// TIA Portal project "Projet_final_groupe_01" (V15.1)

(* hardware
DEVICE "Station S71500/ET200MP_1"  S7-1500 station
   slot 0: "Châssis_0"  Rack  6ES7 590-1***0-0AA0
   slot 1: "PLC_1"  CPU 1513-1 PN  6ES7 513-1AL00-0AB0  V1.7
      slot 3: "Ecran CPU_1"  6ES7591-1AA00-0AA0
   slot 2: "DI 32x24VDC HF_1"  DI 32x24VDC HF  6ES7 521-1BL00-0AB0  V2.0
   slot 3: "DQ 32x24VDC/0.5A ST_1"  DQ 32x24VDC/0.5A ST  6ES7 522-1BL00-0AB0  V2.0
DEVICE "Appareil GSD_1"  GSD.Device.PN
   slot 0: "Châssis"  Rack  V1.0
   slot 0: "PNET-Anybus"  DSQC688  ABCC-PRT  V1.12
      slot 0: "PROFINET Anybus"  PROFINET Anybus  ABCC-PRT  V1.12
      slot 1: "Interface"  Interface
         slot 1: "Port 1"  Port 1
   slot 1: "Input 64 byte_1"  Input 64 byte  V1.0
      slot 0: "Input 64 byte"  Input 64 byte
   slot 2: "Output 64 byte_1"  Output 64 byte  V1.0
      slot 0: "Output 64 byte"  Output 64 byte
DEVICE "Appareil GSD_2"  GSD.Device.PN
   slot 0: "Châssis"  Rack  V1.0
   slot 0: "AL1100"  AL1100  AL1100
      slot 0: "AL1100"  AL1100
      slot 1: "X1"  X1
         slot 1: "Port 1"  Port 1
         slot 2: "Port 2"  Port 2
      slot 1: "4 Ports_1"  4 Ports  AL1100
         slot 0: "IO-Link Master"  IO-Link Master
   slot 1: "IO-Link In  2 Byte + PQI"  IO-Link In  2 Byte + PQI
   slot 2: "Disabled"  Disabled
   slot 3: "Disabled_1"  Disabled
   slot 4: "Disabled_2"  Disabled
*)

// ===== PLC "PLC_1"  CPU 1513-1 PN =====

VAR_GLOBAL   // PLC tag table "Table de variables standard"
   "Sécurité_active" AT %M5.0 : Bool;
   "Marche_cycle" AT %M5.1 : Bool;
   "System_Byte" AT %MB1 : Byte;
   "FirstScan" AT %M1.0 : Bool;
   "DiagStatusUpdate" AT %M1.1 : Bool;
   "AlwaysTRUE" AT %M1.2 : Bool;
   "AlwaysFALSE" AT %M1.3 : Bool;
   "Clock_Byte" AT %MB0 : Byte;
   "Clock_10Hz" AT %M0.0 : Bool;
   "Clock_5Hz" AT %M0.1 : Bool;
   "Clock_2.5Hz" AT %M0.2 : Bool;
   "Clock_2Hz" AT %M0.3 : Bool;
   "Clock_1.25Hz" AT %M0.4 : Bool;
   "Clock_1Hz" AT %M0.5 : Bool;
   "Clock_0.625Hz" AT %M0.6 : Bool;
   "Clock_0.5Hz" AT %M0.7 : Bool;
END_VAR

VAR_GLOBAL   // PLC tag table "Table de variables standard_1"
   "Sécurité_active(1)" AT %M5.0 : Bool;
   "Marche_cycle(1)" AT %M5.1 : Bool;
   "MDM_Local" AT %M5.2 : Bool;
   "MDM_Distant" AT %M5.3 : Bool;
   "MDM_Maintenance" AT %M5.4 : Bool;
   "Demande_arret_propre" AT %M5.5 : Bool;
END_VAR

VAR_GLOBAL CONSTANT   // PLC tag table "Table de variables standard_1"
   "Aucun(e)(1)" : Pip := 65535;
   "Mise à jour automatique(1)" : Pip := 0;
   "MIP 1(1)" : Pip := 1;
   "MIP 2(1)" : Pip := 2;
   "MIP 3(1)" : Pip := 3;
   "MIP 4(1)" : Pip := 4;
   "MIP 5(1)" : Pip := 5;
   "MIP 6(1)" : Pip := 6;
   "MIP 7(1)" : Pip := 7;
   "MIP 8(1)" : Pip := 8;
   "MIP 9(1)" : Pip := 9;
   "MIP 10(1)" : Pip := 10;
   "MIP 11(1)" : Pip := 11;
   "MIP 12(1)" : Pip := 12;
   "MIP 13(1)" : Pip := 13;
   "MIP 14(1)" : Pip := 14;
   "MIP 15(1)" : Pip := 15;
   "MIP 16(1)" : Pip := 16;
   "MIP 17(1)" : Pip := 17;
   "MIP 18(1)" : Pip := 18;
   "MIP 19(1)" : Pip := 19;
   "MIP 20(1)" : Pip := 20;
   "MIP 21(1)" : Pip := 21;
   "MIP 22(1)" : Pip := 22;
   "MIP 23(1)" : Pip := 23;
   "MIP 24(1)" : Pip := 24;
   "MIP 25(1)" : Pip := 25;
   "MIP 26(1)" : Pip := 26;
   "MIP 27(1)" : Pip := 27;
   "MIP 28(1)" : Pip := 28;
   "MIP 29(1)" : Pip := 29;
   "MIP 30(1)" : Pip := 30;
   "MIP 31(1)" : Pip := 31;
   "MIP OB Servo(1)" : Pip := 32768;
   "Local(1)" : Hw_SubModule := 49;
   "Local~Common(1)" : Hw_SubModule := 50;
   "Local~Device(1)" : Hw_Device := 32;
   "Local~Configuration(1)" : Hw_SubModule := 33;
   "Local~Display(1)" : Hw_SubModule := 54;
   "Local~MC(1)" : Hw_SubModule := 51;
   "Local~Exec(1)" : Hw_SubModule := 52;
   "Local~Interface_PROFINET_1(1)" : Hw_Interface := 64;
   "Local~Interface_PROFINET_1~Port_1(1)" : Hw_Interface := 65;
   "Local~Interface_PROFINET_1~Port_2(1)" : Hw_Interface := 66;
   "Local~DI_32x24VDC_HF_1(1)" : Hw_SubModule := 257;
   "Local~DQ_32x24VDC_0_5A_ST_1(1)" : Hw_SubModule := 258;
   "OB_Main(1)" : OB_PCYCLE := 1;
   "Local~PROFINET_IO-System(1)" : Hw_IoSystem := 259;
   "AL1100~Proxy(1)" : Hw_SubModule := 266;
   "AL1100~IODevice(1)" : Hw_Device := 263;
   "AL1100~X1(1)" : Hw_Interface := 267;
   "AL1100~X1~Port_1(1)" : Hw_Interface := 260;
   "AL1100~X1~Port_2(1)" : Hw_Interface := 261;
   "AL1100~Head(1)" : Hw_SubModule := 262;
   "AL1100~4_Ports_1(1)" : Hw_SubModule := 264;
   "PNET-Anybus~Proxy(1)" : Hw_SubModule := 270;
   "PNET-Anybus~IODevice(1)" : Hw_Device := 268;
   "PNET-Anybus~Interface(1)" : Hw_Interface := 271;
   "PNET-Anybus~Interface~Port_1(1)" : Hw_Interface := 272;
   "PNET-Anybus~Head(1)" : Hw_SubModule := 273;
   "PNET-Anybus~Input_64_byte_1(1)" : Hw_SubModule := 274;
   "PNET-Anybus~Output_64_byte_1(1)" : Hw_SubModule := 275;
   "AL1100~4_Ports_1_1(1)" : Hw_SubModule := 276;
   "AL1100~4_Ports_1~IO-Link_In__2_Byte_+_PQI(1)" : Hw_SubModule := 277;
   "AL1100~4_Ports_1~Disabled(1)" : Hw_SubModule := 278;
   "AL1100~4_Ports_1~Disabled_1(1)" : Hw_SubModule := 279;
   "AL1100~4_Ports_1~Disabled_2(1)" : Hw_SubModule := 280;
END_VAR

VAR_GLOBAL   // PLC tag table "Entrées/Sorties"
   "AU_1" AT %I0.0 : Bool;
   "AU_2" AT %I0.1 : Bool;
   "BP_reset" AT %I0.2 : Bool;
   "BP_marche" AT %I0.3 : Bool;
   "BP_arrêt" AT %I0.4 : Bool;
   "Capteur_PP_Assemblage" AT %I1.0 : Bool;
   "Capteur_Distance_brute" AT %IW4 : Word;
   "Motors_ON_INPUT" AT %I100.0 : Bool;
   "Cycle_ON" AT %I100.1 : Bool;
   "Auto_ON" AT %I100.2 : Bool;
   "TCP_SPEED" AT %I100.3 : Bool;
   "Motors_ ON_State" AT %I100.4 : Bool;
   "Task_Executing" AT %I100.5 : Bool;
   "Motors_OFF_INPUT" AT %I100.6 : Bool;
   "Emergency_stop" AT %I100.7 : Bool;
   "Runchain_OK" AT %I101.0 : Bool;
   "Execution_error" AT %I101.1 : Bool;
   "Motors_OFF_State" AT %I101.2 : Bool;
   "Bit_de_vie_robot" AT %I102.0 : Bool;
   "Cycle_en_cours" AT %I106.2 : Bool;
   "Cycle_terminé" AT %I102.3 : Bool;
   "Demande_Offset_prise_pièce_C" AT %I103.0 : Bool;
   "Moteur_convoyeur" AT %Q0.0 : Bool;
   "Motors_ON_OUTPUT" AT %Q100.0 : Bool;
   "Start" AT %Q100.1 : Bool;
   "Stop" AT %Q100.2 : Bool;
   "Soft_stop" AT %Q100.3 : Bool;
   "Interrupt" AT %Q100.4 : Bool;
   "Reset_AU" AT %Q100.5 : Bool;
   "Motors_ON_and_Start" AT %Q100.6 : Bool;
   "Sytem_restart" AT %Q100.7 : Bool;
   "PP_to_Main" AT %Q101.0 : Bool;
   "Motors_OFF_OUTPUT" AT %Q101.1 : Bool;
   "Start_at_Main" AT %Q101.2 : Bool;
   "Quick_Stop" AT %Q101.3 : Bool;
   "Stop_at_end_of_cycle" AT %Q101.4 : Bool;
   "Load_and_start" AT %Q101.5 : Bool;
   "Code_cycle" AT %QW102 : Word;
   "Offset_prise_pièce_C" AT %QW104 : Word;
   "Assemblage_non_conforme" AT %I102.5 : Bool;
   "PP_Assemblage" AT %Q106.3 : Bool;
   "Non_Présence_Pièce_C" AT %I107.5 : Bool;
   "Authorisation_Prise_C" AT %Q106.4 : Bool;
   "Demande_arrêt_propre" AT %Q106.6 : Bool;
   "Position_home" AT %I106.3 : Bool;
   "Etat_de_la_baie" AT %I107.1 : Bool;
   "Voyant_réarmement" AT %Q0.4 : Bool;
   "Voyant_en_cycle" AT %Q0.3 : Bool;
   "Fin_de_prod" AT %I106.4 : Bool;
END_VAR

DATA_BLOCK "DB_Gestion_IHM"   // DB2
{ S7_Optimized_Access := 'FALSE' }
VERSION : 0.1
   VAR
      BP_Init : Bool;
      BP_Home : Bool;
      BP_marche_convoyeur : Bool;
      Capteur_P_assemblage_1 : Bool;
      Mode_Auto : Bool;
      Cycle_en_cours : Bool;
      Sécurité_active : Bool;
      BP_Valider : Bool;
      BP_maintenance : Bool;
      Baie_éteinte : Bool;
      libre_3 : Bool;
      libre_4 : Bool;
      libre_5 : Bool;
      libre_6 : Bool;
      libre_7 : Bool;
      libre_8 : Bool;
      libre_9 : Bool;
      libre_10 : Bool;
      libre_11 : Bool;
      libre_12 : Bool;
      libre_13 : Bool;
      libre_14 : Bool;
      libre_15 : Bool;
      libre_16 : Bool;
      Nombre_palette : Int;
      Mode_de_marche : Int;
      Capteur_distance : Int;
      Code_cycle : Word;
      libre_17 : Int;
      Nombre_palette_distant : Int;
      Fin_de_prod_distant : Int;
      Défaut_Non_Présecence_Pièce_C : Bool;
      Défaut_Présence_Pièce_C_Trop_Haute : Bool;
      "Arrêt_d'urgence" : Bool;
      Robot_pas_en_pos_home : Bool;
      Attente_pièce_assemblage : Bool;
      Test : DInt;
   END_VAR
BEGIN
END_DATA_BLOCK

// folder: System blocks/Program resources

DATA_BLOCK "IEC_Timer_0_DB"   // DB1
{ S7_Optimized_Access := 'TRUE' }
AUTHOR : Simatic
FAMILY : IEC
NAME : IEC_TMR
VERSION : 1.0
// stored: InstanceOfName IEC_TIMER
"IEC_TIMER"
BEGIN
END_DATA_BLOCK

DATA_BLOCK "IEC_Timer_0_DB_1"   // DB3
{ S7_Optimized_Access := 'TRUE' }
AUTHOR : Simatic
FAMILY : IEC
NAME : IEC_TMR
VERSION : 1.0
// stored: InstanceOfName IEC_TIMER
"IEC_TIMER"
BEGIN
END_DATA_BLOCK

// folder: (top level)

FUNCTION "Gestion code cycle" : Void   // FC10, LAD
{ S7_Optimized_Access := 'TRUE' }
VERSION : 0.1
// 100 nb de palette = 1
// 101 = 2
// 102 = 3
// 103 = 4
// 110 Rebus apellé pour mettre une pièce non conforme si la cellule fanuc en done l'ordre et si un appuie sur BP init
// 120 Position home apellé depuis l'IHM
// 130 Position Maintenance appellé depuis IHM
   VAR_TEMP
      Temp_1 : Word;
      Temp_2 : Word;
      Temp_3 : Bool;
      Temp_4 : Bool;
      Temp_5 : Bool;
      Temp_6 : Bool;
      Temp_7 : Bool;
      Temp_8 : Bool;
      Temp_9 : Bool;
   END_VAR
   VAR_TEMP   // added for the SCL form of the ladder/FBD networks
      _w1 : Bool;
   END_VAR
BEGIN

REGION Network 1: Visu voyant cycle en cours IHM
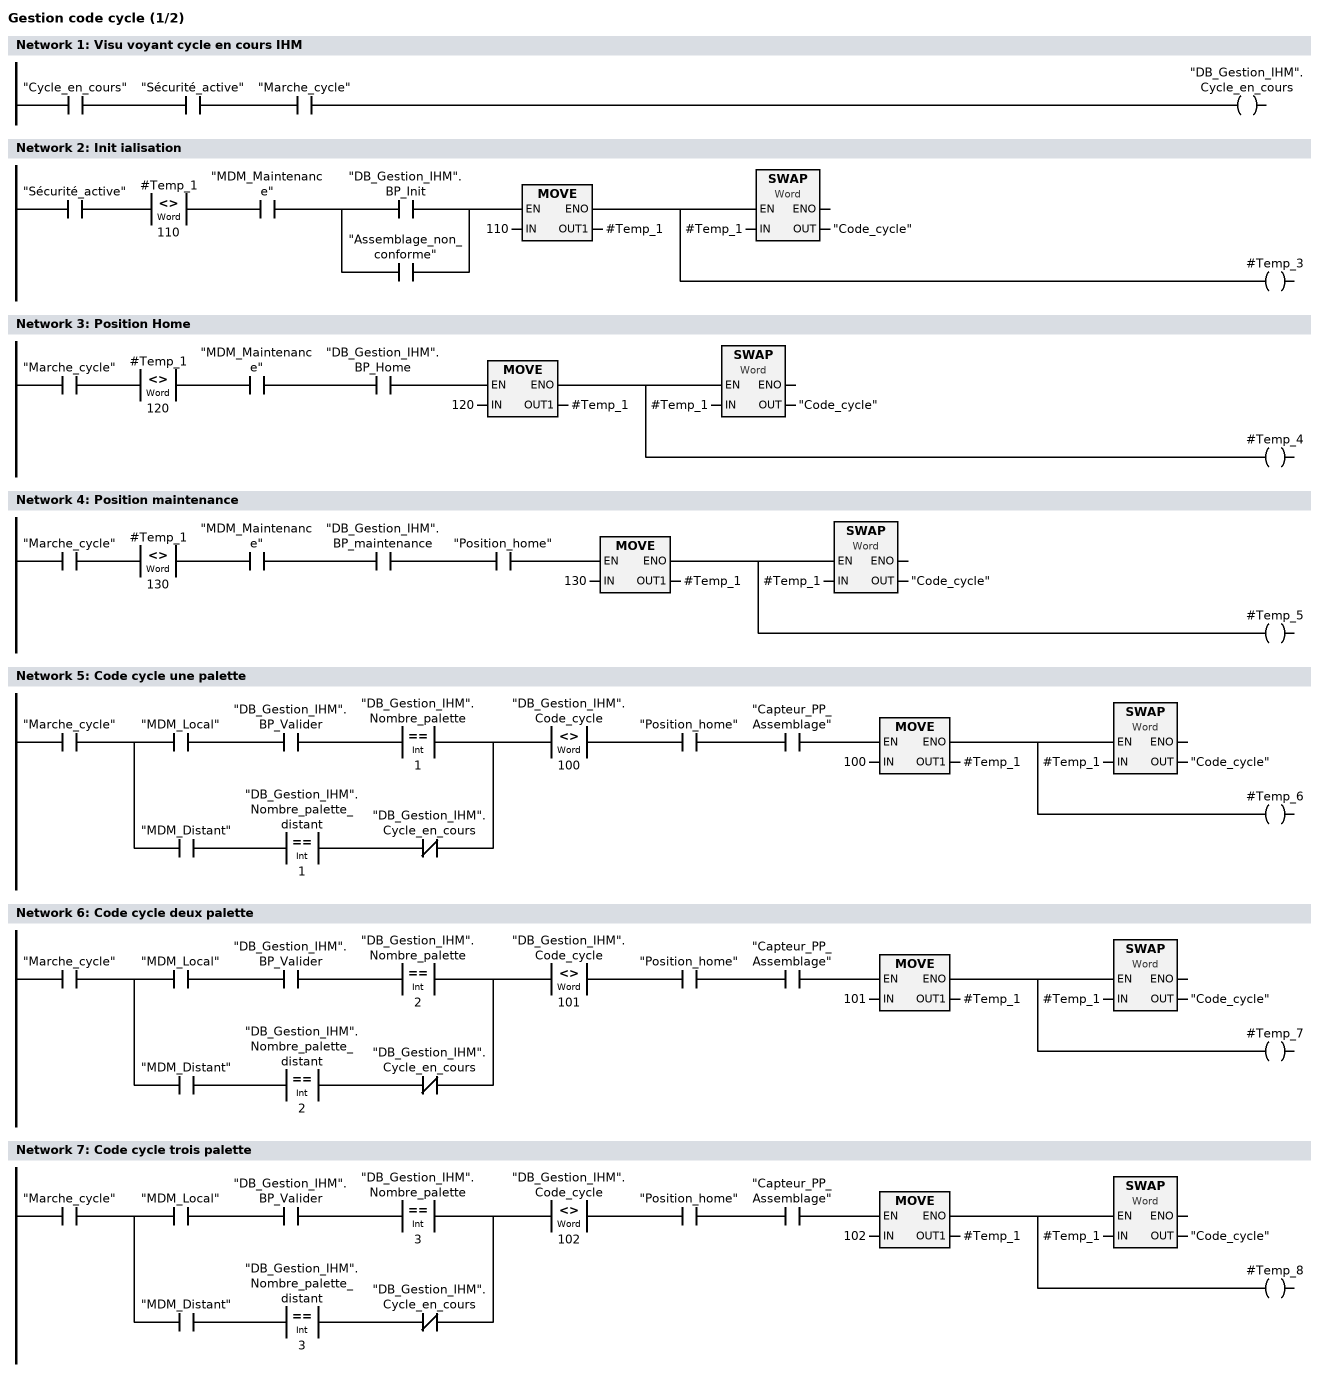
   RUNG wire#powerrail
      Contact( "Cycle_en_cours" )
      Contact( "Sécurité_active" )
      Contact( "Marche_cycle" )
      Coil( "DB_Gestion_IHM".Cycle_en_cours )
   END_RUNG
   // the same network as SCL:
   "DB_Gestion_IHM".Cycle_en_cours := "Cycle_en_cours" AND "Sécurité_active" AND "Marche_cycle";
END_REGION

REGION Network 2: Init ialisation
   #_w1 := "Sécurité_active" AND (#Temp_1 <> 110) AND "MDM_Maintenance" AND ("DB_Gestion_IHM".BP_Init OR "Assemblage_non_conforme");
   IF #_w1 THEN
       #Temp_1 := 110;
       "Code_cycle" := SWAP(#Temp_1);
   END_IF;
   #Temp_3 := #_w1;
END_REGION

REGION Network 3: Position Home
   #_w1 := "Marche_cycle" AND (#Temp_1 <> 120) AND "MDM_Maintenance" AND "DB_Gestion_IHM".BP_Home;
   IF #_w1 THEN
       #Temp_1 := 120;
       "Code_cycle" := SWAP(#Temp_1);
   END_IF;
   #Temp_4 := #_w1;
END_REGION

REGION Network 4: Position maintenance
   #_w1 := "Marche_cycle" AND (#Temp_1 <> 130) AND "MDM_Maintenance" AND "DB_Gestion_IHM".BP_maintenance AND "Position_home";
   IF #_w1 THEN
       #Temp_1 := 130;
       "Code_cycle" := SWAP(#Temp_1);
   END_IF;
   #Temp_5 := #_w1;
END_REGION

REGION Network 5: Code cycle une palette
   #_w1 := "Marche_cycle" AND (("MDM_Local" AND "DB_Gestion_IHM".BP_Valider AND ("DB_Gestion_IHM".Nombre_palette = 1)) OR ("MDM_Distant" AND ("DB_Gestion_IHM".Nombre_palette_distant = 1) AND NOT "DB_Gestion_IHM".Cycle_en_cours)) AND ("DB_Gestion_IHM".Code_cycle <> 100) AND "Position_home" AND "Capteur_PP_Assemblage";
   IF #_w1 THEN
       #Temp_1 := 100;
       "Code_cycle" := SWAP(#Temp_1);
   END_IF;
   #Temp_6 := #_w1;
END_REGION

REGION Network 6: Code cycle deux palette
   #_w1 := "Marche_cycle" AND (("MDM_Local" AND "DB_Gestion_IHM".BP_Valider AND ("DB_Gestion_IHM".Nombre_palette = 2)) OR ("MDM_Distant" AND ("DB_Gestion_IHM".Nombre_palette_distant = 2) AND NOT "DB_Gestion_IHM".Cycle_en_cours)) AND ("DB_Gestion_IHM".Code_cycle <> 101) AND "Position_home" AND "Capteur_PP_Assemblage";
   IF #_w1 THEN
       #Temp_1 := 101;
       "Code_cycle" := SWAP(#Temp_1);
   END_IF;
   #Temp_7 := #_w1;
END_REGION

REGION Network 7: Code cycle trois palette
   #_w1 := "Marche_cycle" AND (("MDM_Local" AND "DB_Gestion_IHM".BP_Valider AND ("DB_Gestion_IHM".Nombre_palette = 3)) OR ("MDM_Distant" AND ("DB_Gestion_IHM".Nombre_palette_distant = 3) AND NOT "DB_Gestion_IHM".Cycle_en_cours)) AND ("DB_Gestion_IHM".Code_cycle <> 102) AND "Position_home" AND "Capteur_PP_Assemblage";
   IF #_w1 THEN
       #Temp_1 := 102;
       "Code_cycle" := SWAP(#Temp_1);
   END_IF;
   #Temp_8 := #_w1;
END_REGION

REGION Network 8: Code cycle quatre palette
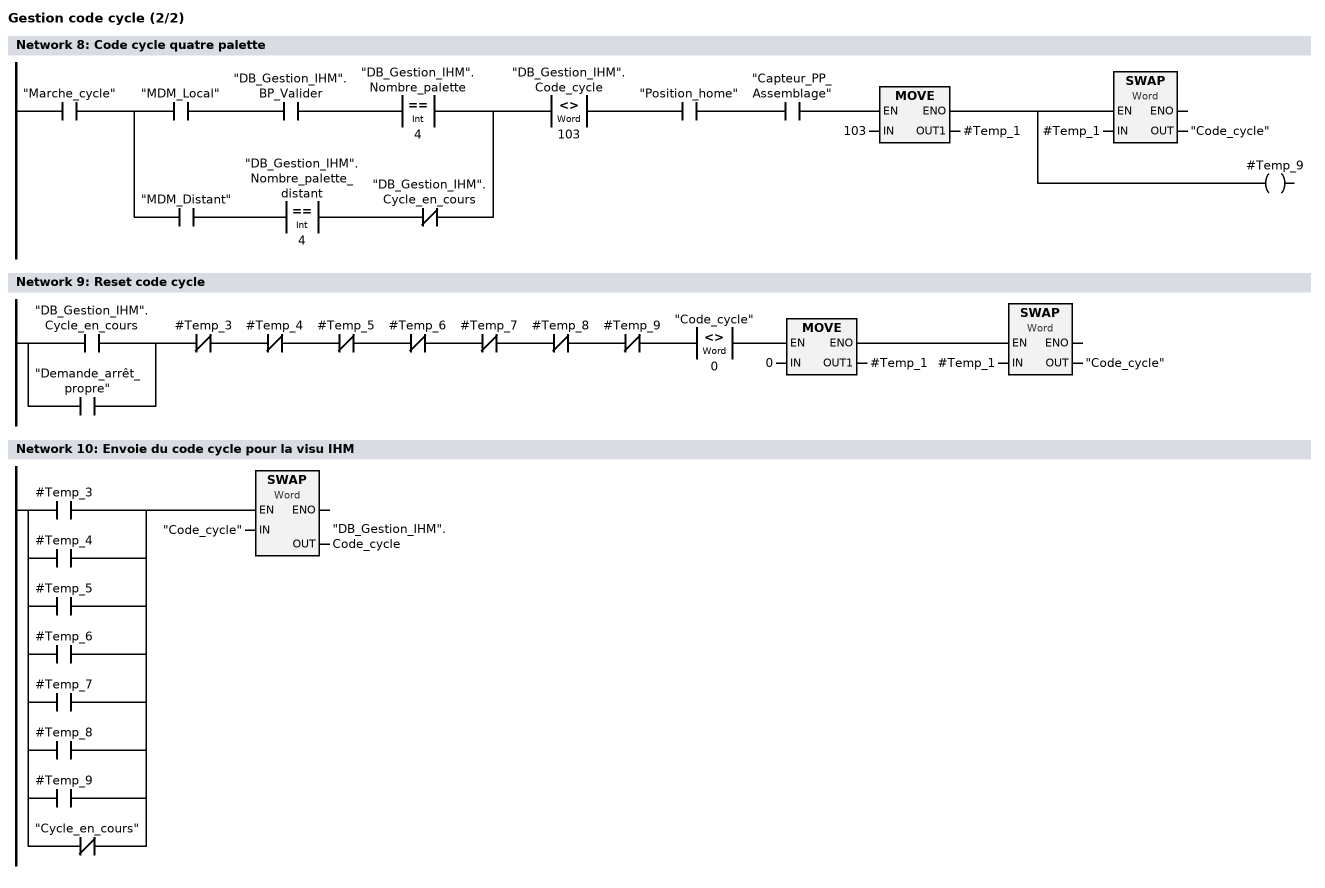
   #_w1 := "Marche_cycle" AND (("MDM_Local" AND "DB_Gestion_IHM".BP_Valider AND ("DB_Gestion_IHM".Nombre_palette = 4)) OR ("MDM_Distant" AND ("DB_Gestion_IHM".Nombre_palette_distant = 4) AND NOT "DB_Gestion_IHM".Cycle_en_cours)) AND ("DB_Gestion_IHM".Code_cycle <> 103) AND "Position_home" AND "Capteur_PP_Assemblage";
   IF #_w1 THEN
       #Temp_1 := 103;
       "Code_cycle" := SWAP(#Temp_1);
   END_IF;
   #Temp_9 := #_w1;
END_REGION

REGION Network 9: Reset code cycle
   IF ("DB_Gestion_IHM".Cycle_en_cours OR "Demande_arrêt_propre") AND NOT #Temp_3 AND NOT #Temp_4 AND NOT #Temp_5 AND NOT #Temp_6 AND NOT #Temp_7 AND NOT #Temp_8 AND NOT #Temp_9 AND ("Code_cycle" <> 0) THEN
       #Temp_1 := 0;
       "Code_cycle" := SWAP(#Temp_1);
   END_IF;
END_REGION

REGION Network 10: Envoie du code cycle pour la visu IHM
   IF #Temp_3 OR #Temp_4 OR #Temp_5 OR #Temp_6 OR #Temp_7 OR #Temp_8 OR #Temp_9 OR NOT "Cycle_en_cours" THEN
       "DB_Gestion_IHM".Code_cycle := SWAP("Code_cycle");
   END_IF;
END_REGION
END_FUNCTION

FUNCTION "Gestion marche cellule" : Void   // FC11, LAD
{ S7_Optimized_Access := 'TRUE' }
VERSION : 0.1
   VAR_TEMP   // added for the SCL form of the ladder/FBD networks
      _w1 : Bool;
   END_VAR
BEGIN

REGION Network 1: Marche cycle et Moteurs à ON
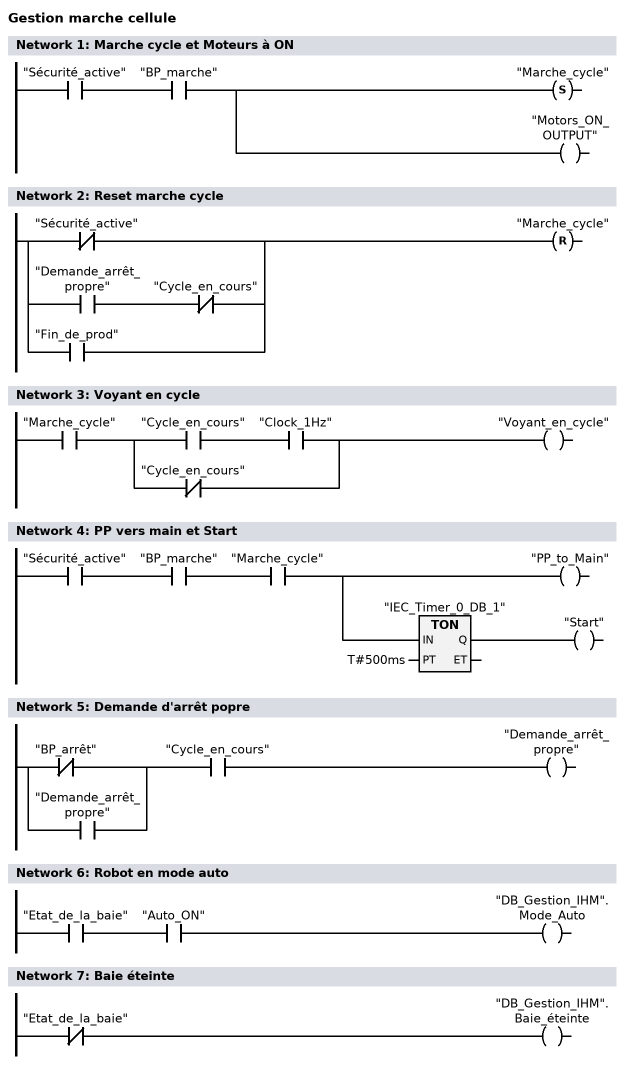
   RUNG wire#powerrail
      Contact( "Sécurité_active" )
      Contact( "BP_marche" )
      wire#w1
      S_Coil( "Marche_cycle" )
   END_RUNG
   RUNG wire#w1
      Coil( "Motors_ON_OUTPUT" )
   END_RUNG
   // the same network as SCL:
   #_w1 := "Sécurité_active" AND "BP_marche";
   IF #_w1 THEN "Marche_cycle" := TRUE; END_IF;
   "Motors_ON_OUTPUT" := #_w1;
END_REGION

REGION Network 2: Reset marche cycle
   RUNG wire#powerrail
      I_Contact( "Sécurité_active" )
      wire#w1
      R_Coil( "Marche_cycle" )
   END_RUNG
   RUNG wire#powerrail
      Contact( "Demande_arrêt_propre" )
      I_Contact( "Cycle_en_cours" )
   END_RUNG wire#w1
   RUNG wire#powerrail
      Contact( "Fin_de_prod" )
   END_RUNG wire#w1
   // the same network as SCL:
   IF NOT "Sécurité_active" OR ("Demande_arrêt_propre" AND NOT "Cycle_en_cours") OR "Fin_de_prod" THEN
       "Marche_cycle" := FALSE;
   END_IF;
END_REGION

REGION Network 3: Voyant en cycle
   RUNG wire#powerrail
      Contact( "Marche_cycle" )
      wire#w1
      Contact( "Cycle_en_cours" )
      Contact( "Clock_1Hz" )
      wire#w2
      Coil( "Voyant_en_cycle" )
   END_RUNG
   RUNG wire#w1
      I_Contact( "Cycle_en_cours" )
   END_RUNG wire#w2
   // the same network as SCL:
   "Voyant_en_cycle" := "Marche_cycle" AND (("Cycle_en_cours" AND "Clock_1Hz") OR NOT "Cycle_en_cours");
END_REGION

REGION Network 4: PP vers main et Start
   "PP_to_Main" := "Sécurité_active" AND "BP_marche" AND "Marche_cycle";
   "IEC_Timer_0_DB_1".TON(IN := "PP_to_Main", PT := T#500ms);
   "Start" := "IEC_Timer_0_DB_1".Q;
END_REGION

REGION Network 5: Demande d'arrêt popre
   RUNG wire#powerrail
      I_Contact( "BP_arrêt" )
      wire#w1
      Contact( "Cycle_en_cours" )
      Coil( "Demande_arrêt_propre" )
   END_RUNG
   RUNG wire#powerrail
      Contact( "Demande_arrêt_propre" )
   END_RUNG wire#w1
   // the same network as SCL:
   "Demande_arrêt_propre" := (NOT "BP_arrêt" OR "Demande_arrêt_propre") AND "Cycle_en_cours";
END_REGION

REGION Network 6: Robot en mode auto
   RUNG wire#powerrail
      Contact( "Etat_de_la_baie" )
      Contact( "Auto_ON" )
      Coil( "DB_Gestion_IHM".Mode_Auto )
   END_RUNG
   // the same network as SCL:
   "DB_Gestion_IHM".Mode_Auto := "Etat_de_la_baie" AND "Auto_ON";
END_REGION

REGION Network 7: Baie éteinte
   RUNG wire#powerrail
      I_Contact( "Etat_de_la_baie" )
      Coil( "DB_Gestion_IHM".Baie_éteinte )
   END_RUNG
   // the same network as SCL:
   "DB_Gestion_IHM".Baie_éteinte := NOT "Etat_de_la_baie";
END_REGION
END_FUNCTION

FUNCTION "Gestion convoyeur" : Void   // FC12, LAD
{ S7_Optimized_Access := 'TRUE' }
VERSION : 0.1
BEGIN

REGION Network 1: Marche moteur convoyeur
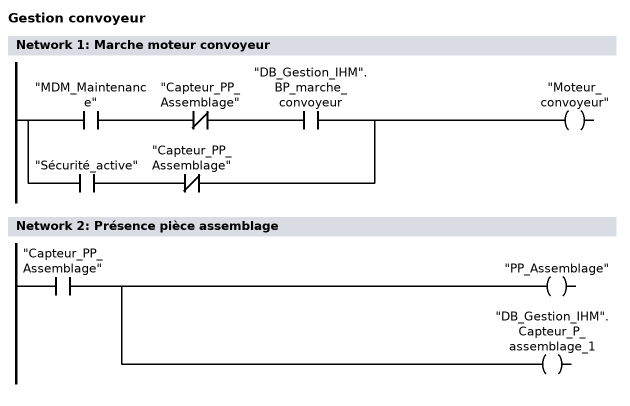
   RUNG wire#powerrail
      Contact( "MDM_Maintenance" )
      I_Contact( "Capteur_PP_Assemblage" )
      Contact( "DB_Gestion_IHM".BP_marche_convoyeur )
      wire#w1
      Coil( "Moteur_convoyeur" )
   END_RUNG
   RUNG wire#powerrail
      Contact( "Sécurité_active" )
      I_Contact( "Capteur_PP_Assemblage" )
   END_RUNG wire#w1
   // the same network as SCL:
   "Moteur_convoyeur" := ("MDM_Maintenance" AND NOT "Capteur_PP_Assemblage" AND "DB_Gestion_IHM".BP_marche_convoyeur) OR ("Sécurité_active" AND NOT "Capteur_PP_Assemblage");
END_REGION

REGION Network 2: Présence pièce assemblage
   RUNG wire#powerrail
      Contact( "Capteur_PP_Assemblage" )
      wire#w1
      Coil( "PP_Assemblage" )
   END_RUNG
   RUNG wire#w1
      Coil( "DB_Gestion_IHM".Capteur_P_assemblage_1 )
   END_RUNG
   // the same network as SCL:
   "PP_Assemblage" := "Capteur_PP_Assemblage";
   "DB_Gestion_IHM".Capteur_P_assemblage_1 := "Capteur_PP_Assemblage";
END_REGION
END_FUNCTION

FUNCTION "Gestion mode de marche" : Void   // FC13, LAD
{ S7_Optimized_Access := 'TRUE' }
VERSION : 0.1
BEGIN

REGION Network 1: Mode de marche local
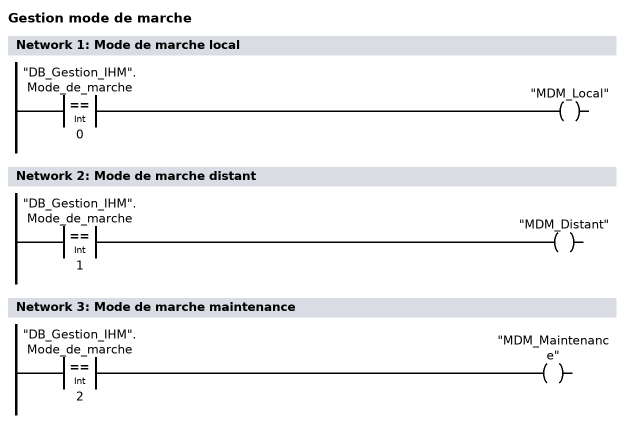
   RUNG wire#powerrail
      { S7_Templates := "SrcType := Int" } EQ_Contact(in1 := "DB_Gestion_IHM".Mode_de_marche, in2 := 0)
      Coil( "MDM_Local" )
   END_RUNG
   // the same network as SCL:
   "MDM_Local" := "DB_Gestion_IHM".Mode_de_marche = 0;
END_REGION

REGION Network 2: Mode de marche distant
   RUNG wire#powerrail
      { S7_Templates := "SrcType := Int" } EQ_Contact(in1 := "DB_Gestion_IHM".Mode_de_marche, in2 := 1)
      Coil( "MDM_Distant" )
   END_RUNG
   // the same network as SCL:
   "MDM_Distant" := "DB_Gestion_IHM".Mode_de_marche = 1;
END_REGION

REGION Network 3: Mode de marche maintenance
   RUNG wire#powerrail
      { S7_Templates := "SrcType := Int" } EQ_Contact(in1 := "DB_Gestion_IHM".Mode_de_marche, in2 := 2)
      Coil( "MDM_Maintenance" )
   END_RUNG
   // the same network as SCL:
   "MDM_Maintenance" := "DB_Gestion_IHM".Mode_de_marche = 2;
END_REGION
END_FUNCTION

FUNCTION "Mode de marche distant" : Void   // FC20, LAD
{ S7_Optimized_Access := 'TRUE' }
VERSION : 0.1
   VAR_TEMP
      temp_1 : Bool;
   END_VAR
BEGIN

REGION Network 1: Fin de prod pour cloturer l'OF
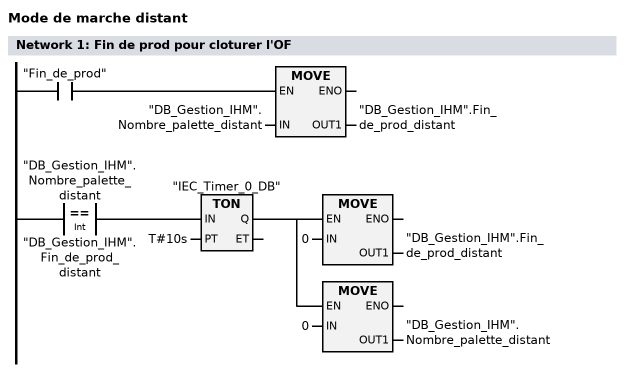
   IF "Fin_de_prod" THEN
       "DB_Gestion_IHM".Fin_de_prod_distant := "DB_Gestion_IHM".Nombre_palette_distant;
   END_IF;
   "IEC_Timer_0_DB".TON(IN := "DB_Gestion_IHM".Nombre_palette_distant = "DB_Gestion_IHM".Fin_de_prod_distant,
                        PT := T#10s);
   IF "IEC_Timer_0_DB".Q THEN
       "DB_Gestion_IHM".Fin_de_prod_distant := 0;
       "DB_Gestion_IHM".Nombre_palette_distant := 0;
   END_IF;
END_REGION
END_FUNCTION

FUNCTION "Gestion Alarme IHM" : Void   // FC30, LAD
{ S7_Optimized_Access := 'TRUE' }
VERSION : 0.1
BEGIN

REGION Network 1: Erreur pas en position home
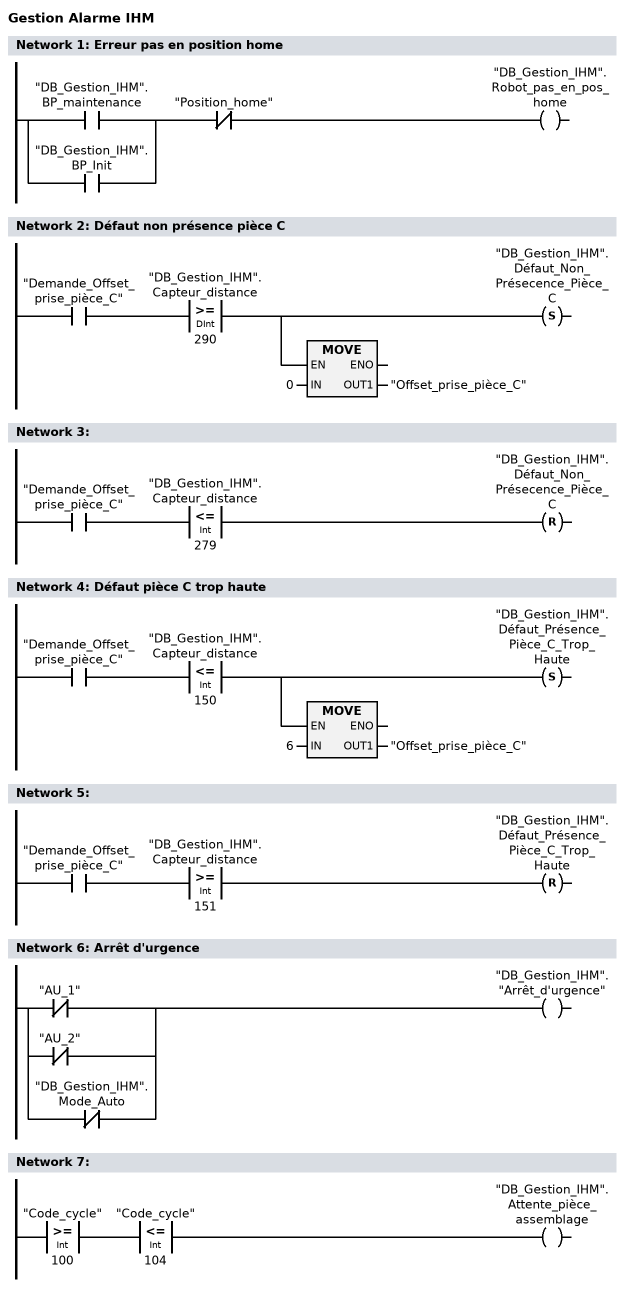
   RUNG wire#powerrail
      Contact( "DB_Gestion_IHM".BP_maintenance )
      wire#w1
      I_Contact( "Position_home" )
      Coil( "DB_Gestion_IHM".Robot_pas_en_pos_home )
   END_RUNG
   RUNG wire#powerrail
      Contact( "DB_Gestion_IHM".BP_Init )
   END_RUNG wire#w1
   // the same network as SCL:
   "DB_Gestion_IHM".Robot_pas_en_pos_home := ("DB_Gestion_IHM".BP_maintenance OR "DB_Gestion_IHM".BP_Init) AND NOT "Position_home";
END_REGION

REGION Network 2: Défaut non présence pièce C
   RUNG wire#powerrail
      Contact( "Demande_Offset_prise_pièce_C" )
      { S7_Templates := "SrcType := DInt" } GE_Contact(in1 := "DB_Gestion_IHM".Capteur_distance, in2 := 290)
      wire#w1
      S_Coil( "DB_Gestion_IHM".Défaut_Non_Présecence_Pièce_C )
   END_RUNG
   RUNG wire#w1
      Move(in := 0, out1 => "Offset_prise_pièce_C")
   END_RUNG
   // the same network as SCL:
   IF "Demande_Offset_prise_pièce_C" AND ("DB_Gestion_IHM".Capteur_distance >= 290) THEN
       "DB_Gestion_IHM".Défaut_Non_Présecence_Pièce_C := TRUE;
       "Offset_prise_pièce_C" := 0;
   END_IF;
END_REGION

REGION Network 3
   RUNG wire#powerrail
      Contact( "Demande_Offset_prise_pièce_C" )
      { S7_Templates := "SrcType := Int" } LE_Contact(in1 := "DB_Gestion_IHM".Capteur_distance, in2 := 279)
      R_Coil( "DB_Gestion_IHM".Défaut_Non_Présecence_Pièce_C )
   END_RUNG
   // the same network as SCL:
   IF "Demande_Offset_prise_pièce_C" AND ("DB_Gestion_IHM".Capteur_distance <= 279) THEN
       "DB_Gestion_IHM".Défaut_Non_Présecence_Pièce_C := FALSE;
   END_IF;
END_REGION

REGION Network 4: Défaut pièce C trop haute
   RUNG wire#powerrail
      Contact( "Demande_Offset_prise_pièce_C" )
      { S7_Templates := "SrcType := Int" } LE_Contact(in1 := "DB_Gestion_IHM".Capteur_distance, in2 := 150)
      wire#w1
      S_Coil( "DB_Gestion_IHM".Défaut_Présence_Pièce_C_Trop_Haute )
   END_RUNG
   RUNG wire#w1
      Move(in := 6, out1 => "Offset_prise_pièce_C")
   END_RUNG
   // the same network as SCL:
   IF "Demande_Offset_prise_pièce_C" AND ("DB_Gestion_IHM".Capteur_distance <= 150) THEN
       "DB_Gestion_IHM".Défaut_Présence_Pièce_C_Trop_Haute := TRUE;
       "Offset_prise_pièce_C" := 6;
   END_IF;
END_REGION

REGION Network 5
   RUNG wire#powerrail
      Contact( "Demande_Offset_prise_pièce_C" )
      { S7_Templates := "SrcType := Int" } GE_Contact(in1 := "DB_Gestion_IHM".Capteur_distance, in2 := 151)
      R_Coil( "DB_Gestion_IHM".Défaut_Présence_Pièce_C_Trop_Haute )
   END_RUNG
   // the same network as SCL:
   IF "Demande_Offset_prise_pièce_C" AND ("DB_Gestion_IHM".Capteur_distance >= 151) THEN
       "DB_Gestion_IHM".Défaut_Présence_Pièce_C_Trop_Haute := FALSE;
   END_IF;
END_REGION

REGION Network 6: Arrêt d'urgence
   RUNG wire#powerrail
      I_Contact( "AU_1" )
      wire#w1
      Coil( "DB_Gestion_IHM"."Arrêt_d'urgence" )
   END_RUNG
   RUNG wire#powerrail
      I_Contact( "AU_2" )
   END_RUNG wire#w1
   RUNG wire#powerrail
      I_Contact( "DB_Gestion_IHM".Mode_Auto )
   END_RUNG wire#w1
   // the same network as SCL:
   "DB_Gestion_IHM"."Arrêt_d'urgence" := NOT "AU_1" OR NOT "AU_2" OR NOT "DB_Gestion_IHM".Mode_Auto;
END_REGION

REGION Network 7
   RUNG wire#powerrail
      { S7_Templates := "SrcType := Int" } GE_Contact(in1 := "Code_cycle", in2 := 100)
      { S7_Templates := "SrcType := Int" } LE_Contact(in1 := "Code_cycle", in2 := 104)
      Coil( "DB_Gestion_IHM".Attente_pièce_assemblage )
   END_RUNG
   // the same network as SCL:
   "DB_Gestion_IHM".Attente_pièce_assemblage := ("Code_cycle" >= 100) AND ("Code_cycle" <= 104);
END_REGION
END_FUNCTION

FUNCTION "Gestion capteurs distance" : Void   // FC70, LAD
{ S7_Optimized_Access := 'TRUE' }
VERSION : 0.1
   VAR_TEMP
      Temp_1 : Real;
      Temp_3 : DWord;
      Temp_2 : Word;
      Temp_4 : Int;
   END_VAR
BEGIN

REGION Network 1: Mise à l'échelle
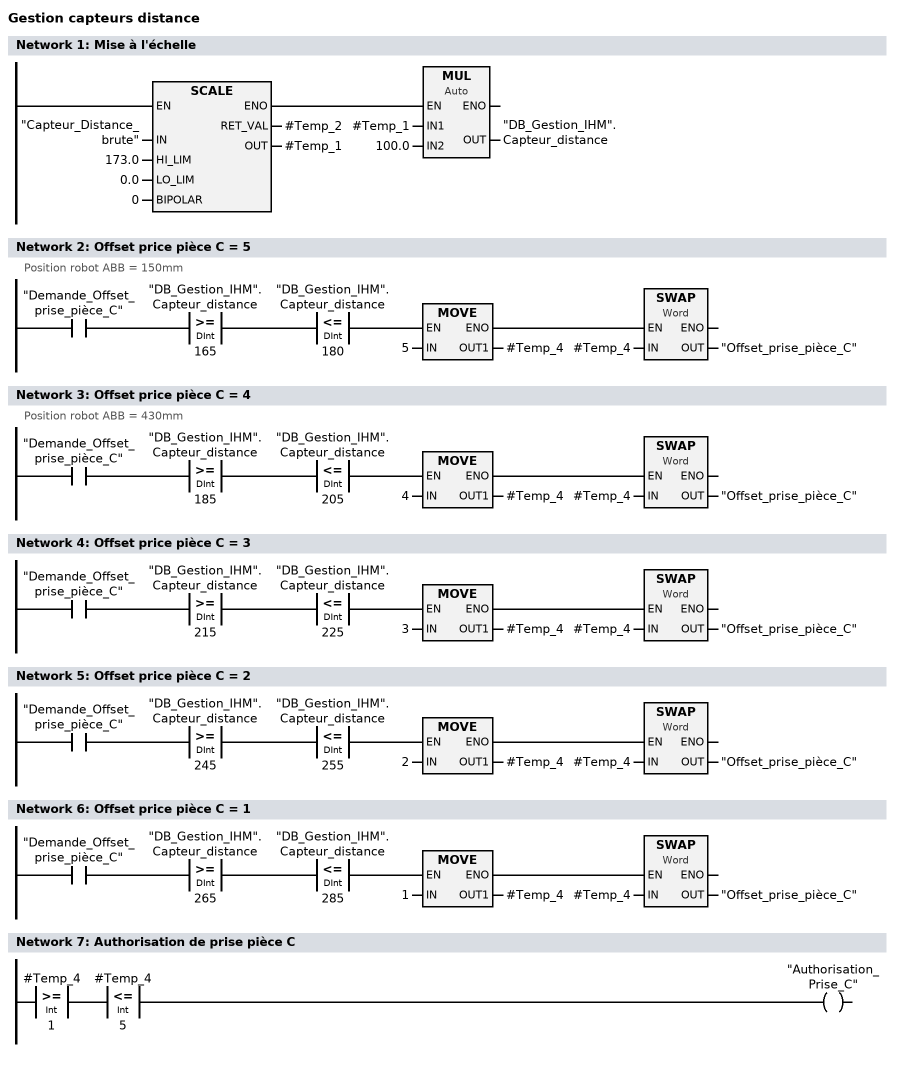
   // ENO of a box is taken as its EN; it also drops when the box reports an error
   #Temp_2 := SCALE(IN := "Capteur_Distance_brute",
                    HI_LIM := 173.0,
                    LO_LIM := 0.0,
                    BIPOLAR := 0,
                    OUT => #Temp_1);
   "DB_Gestion_IHM".Capteur_distance := #Temp_1 * 100.0;
END_REGION

REGION Network 2: Offset price pièce C = 5
   // Position robot ABB = 150mm
   IF "Demande_Offset_prise_pièce_C" AND ("DB_Gestion_IHM".Capteur_distance >= 165) AND ("DB_Gestion_IHM".Capteur_distance <= 180) THEN
       #Temp_4 := 5;
       "Offset_prise_pièce_C" := SWAP(#Temp_4);
   END_IF;
END_REGION

REGION Network 3: Offset price pièce C = 4
   // Position robot ABB = 430mm
   IF "Demande_Offset_prise_pièce_C" AND ("DB_Gestion_IHM".Capteur_distance >= 185) AND ("DB_Gestion_IHM".Capteur_distance <= 205) THEN
       #Temp_4 := 4;
       "Offset_prise_pièce_C" := SWAP(#Temp_4);
   END_IF;
END_REGION

REGION Network 4: Offset price pièce C = 3
   IF "Demande_Offset_prise_pièce_C" AND ("DB_Gestion_IHM".Capteur_distance >= 215) AND ("DB_Gestion_IHM".Capteur_distance <= 225) THEN
       #Temp_4 := 3;
       "Offset_prise_pièce_C" := SWAP(#Temp_4);
   END_IF;
END_REGION

REGION Network 5: Offset price pièce C = 2
   IF "Demande_Offset_prise_pièce_C" AND ("DB_Gestion_IHM".Capteur_distance >= 245) AND ("DB_Gestion_IHM".Capteur_distance <= 255) THEN
       #Temp_4 := 2;
       "Offset_prise_pièce_C" := SWAP(#Temp_4);
   END_IF;
END_REGION

REGION Network 6: Offset price pièce C = 1
   IF "Demande_Offset_prise_pièce_C" AND ("DB_Gestion_IHM".Capteur_distance >= 265) AND ("DB_Gestion_IHM".Capteur_distance <= 285) THEN
       #Temp_4 := 1;
       "Offset_prise_pièce_C" := SWAP(#Temp_4);
   END_IF;
END_REGION

REGION Network 7: Authorisation de prise pièce C
   RUNG wire#powerrail
      { S7_Templates := "SrcType := Int" } GE_Contact(in1 := #Temp_4, in2 := 1)
      { S7_Templates := "SrcType := Int" } LE_Contact(in1 := #Temp_4, in2 := 5)
      Coil( "Authorisation_Prise_C" )
   END_RUNG
   // the same network as SCL:
   "Authorisation_Prise_C" := (#Temp_4 >= 1) AND (#Temp_4 <= 5);
END_REGION
END_FUNCTION

FUNCTION "Sécurité" : Void   // FC100, LAD
{ S7_Optimized_Access := 'TRUE' }
VERSION : 0.1
   VAR_TEMP   // added for the SCL form of the ladder/FBD networks
      _w1 : Bool;
   END_VAR
BEGIN

REGION Network 1
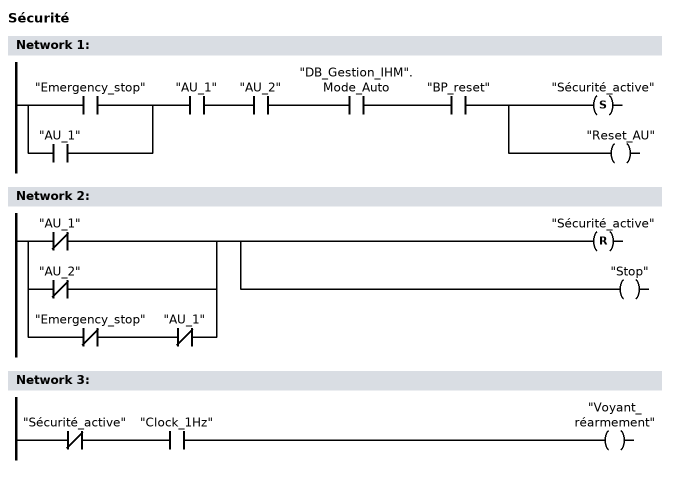
   RUNG wire#powerrail
      Contact( "Emergency_stop" )
      wire#w1
      Contact( "AU_1" )
      Contact( "AU_2" )
      Contact( "DB_Gestion_IHM".Mode_Auto )
      Contact( "BP_reset" )
      wire#w2
      S_Coil( "Sécurité_active" )
   END_RUNG
   RUNG wire#powerrail
      Contact( "AU_1" )
   END_RUNG wire#w1
   RUNG wire#w2
      Coil( "Reset_AU" )
   END_RUNG
   // the same network as SCL:
   #_w1 := ("Emergency_stop" OR "AU_1") AND "AU_1" AND "AU_2" AND "DB_Gestion_IHM".Mode_Auto AND "BP_reset";
   IF #_w1 THEN "Sécurité_active" := TRUE; END_IF;
   "Reset_AU" := #_w1;
END_REGION

REGION Network 2
   RUNG wire#powerrail
      I_Contact( "AU_1" )
      wire#w1
      R_Coil( "Sécurité_active" )
   END_RUNG
   RUNG wire#powerrail
      I_Contact( "AU_2" )
   END_RUNG wire#w1
   RUNG wire#powerrail
      I_Contact( "Emergency_stop" )
      I_Contact( "AU_1" )
   END_RUNG wire#w1
   RUNG wire#w1
      Coil( "Stop" )
   END_RUNG
   // the same network as SCL:
   #_w1 := NOT "AU_1" OR NOT "AU_2" OR (NOT "Emergency_stop" AND NOT "AU_1");
   IF #_w1 THEN "Sécurité_active" := FALSE; END_IF;
   "Stop" := #_w1;
END_REGION

REGION Network 3
   RUNG wire#powerrail
      I_Contact( "Sécurité_active" )
      Contact( "Clock_1Hz" )
      Coil( "Voyant_réarmement" )
   END_RUNG
   // the same network as SCL:
   "Voyant_réarmement" := NOT "Sécurité_active" AND "Clock_1Hz";
END_REGION
END_FUNCTION

ORGANIZATION_BLOCK "Main"   // OB1, LAD, ProgramCycle
TITLE = "Main Program Sweep (Cycle)"
{ S7_Optimized_Access := 'TRUE' }
VERSION : 0.1
   VAR_INPUT
      Initial_Call : Bool;   // Initial call of this OB
      Remanence : Bool;   // =True, if remanent data are available
   END_VAR
BEGIN

REGION Network 1
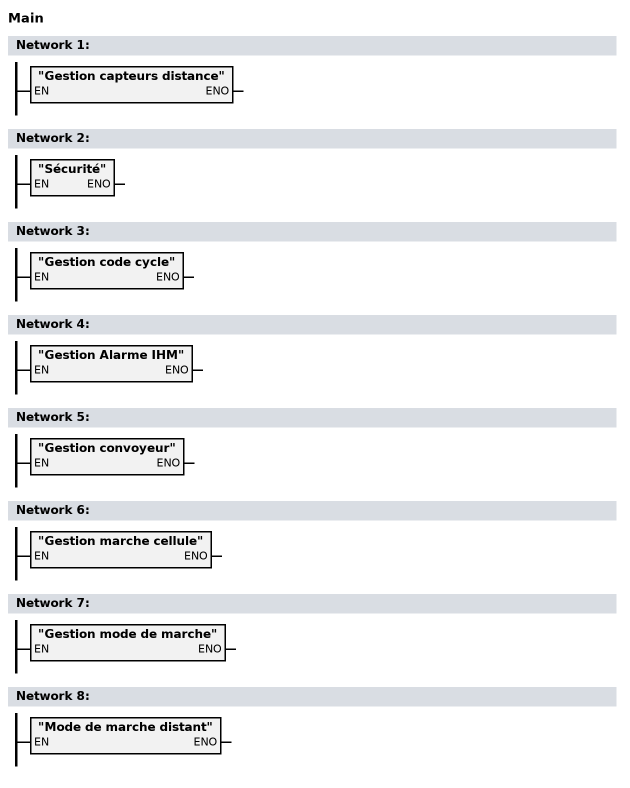
   RUNG wire#powerrail
      "Gestion capteurs distance"()
   END_RUNG
   // the same network as SCL:
   "Gestion capteurs distance"();
END_REGION

REGION Network 2
   RUNG wire#powerrail
      "Sécurité"()
   END_RUNG
   // the same network as SCL:
   "Sécurité"();
END_REGION

REGION Network 3
   RUNG wire#powerrail
      "Gestion code cycle"()
   END_RUNG
   // the same network as SCL:
   "Gestion code cycle"();
END_REGION

REGION Network 4
   RUNG wire#powerrail
      "Gestion Alarme IHM"()
   END_RUNG
   // the same network as SCL:
   "Gestion Alarme IHM"();
END_REGION

REGION Network 5
   RUNG wire#powerrail
      "Gestion convoyeur"()
   END_RUNG
   // the same network as SCL:
   "Gestion convoyeur"();
END_REGION

REGION Network 6
   RUNG wire#powerrail
      "Gestion marche cellule"()
   END_RUNG
   // the same network as SCL:
   "Gestion marche cellule"();
END_REGION

REGION Network 7
   RUNG wire#powerrail
      "Gestion mode de marche"()
   END_RUNG
   // the same network as SCL:
   "Gestion mode de marche"();
END_REGION

REGION Network 8
   RUNG wire#powerrail
      "Mode de marche distant"()
   END_RUNG
   // the same network as SCL:
   "Mode de marche distant"();
END_REGION
END_ORGANIZATION_BLOCK